// TwinCAT 3 PLC project RetentiveTimers
// Title: Retentive Timers
// Company: FisoThemes
// Author: Goodwill Mzumala
// ProjectVersion: 0.1.0.0
// Description: Standard library timers on TwinCAT count time by taking the difference between the current time from system timer and start time from system timer. While this is fine for most application, it is problematic for operations that require time to be retained even if the PLC is paused, stopped or turned off. For example, if a `TON` (Timer On-Delay) Timer is running and you stop the PLC Boot Project for a period of time, the `TON` will not resume from the point it was stopped. Instead it will skip time by the number of ms/secs/mins/hours it was stopped. This makes it useless for applications such as tracking the length of time a PLC has been running or retaining persistent time. Retentive variants of the Standard library timers stop this from happen. They are based on PLC Task cycle time rather than system time. This means they will simply stop counting when the PLC Task Cycle is stopped and will resume from where they left-off as soon as the task cycle picks up. All arguments behave in the same manner as those of the standard library.
// ProgramVersion: 3.1.4023.0
// libraries:
//   Tc2_Standard, * (Beckhoff Automation GmbH)
//   Tc2_System, * (Beckhoff Automation GmbH)
//   Tc3_Module, * (Beckhoff Automation GmbH)
// project tree:
//   DUTs/Structs/ ST_PLC_TASK_INFORMATION.TcDUT
//   / PlcTask.TcTTO
//   POUs/Examples/Section 1 - Standard Timers Comparisons/ P_Example_3_TPs.TcPOU, P_Section_1.TcPOU, P_Example_1_TONs.TcPOU, P_Example_2_TOFs.TcPOU
//   POUs/Examples/Section 2 - Pausable Timers Comparisons/ P_Section_2.TcPOU
//   POUs/Examples/Section 3 - Stopwatch/ P_Example_Stopwatch.TcPOU, P_Section_3.TcPOU
//   POUs/Function Blocks/ FB_RTimer.TcPOU, FB_RTON.TcPOU, FB_RTOF.TcPOU, FB_RTP.TcPOU, FB_RStopwatch.TcPOU, FB_Timer.TcPOU, FB_Stopwatch.TcPOU
//   POUs/Functions/ F_Get_PLC_Task_Information.TcPOU
//   POUs/ MAIN.TcPOU
// real-time tasks:
//   TASK PlcTask: cycle T#10ms, priority 20, ADS port 350

CONFIGURATION RetentiveTimers
    RESOURCE PLC ON TwinCAT3
        TASK PlcTask(INTERVAL := T#10ms, PRIORITY := 20);
        PROGRAM MAIN WITH PlcTask : MAIN;
    END_RESOURCE
END_CONFIGURATION

// ---- DUTs/Structs/ST_PLC_TASK_INFORMATION.TcDUT
TYPE ST_PLC_TASK_INFORMATION EXTENDS PlcTaskSystemInfo :
STRUCT
	tCycleTime 	: TIME; 	// Current task cycle time
	tlCycleTime : LTIME; 	// Current task cycle time in LTIME
END_STRUCT
END_TYPE

// ---- POUs/MAIN.TcPOU
PROGRAM MAIN
VAR
END_VAR

P_Section_1();
P_Section_2();
P_Section_3();

END_PROGRAM

// ---- POUs/Examples/Section 1 - Standard Timers Comparisons/P_Section_1.TcPOU
PROGRAM P_Section_1
VAR
END_VAR

P_Example_1_TONs();
P_Example_2_TOFs();
P_Example_3_TPs();

END_PROGRAM

// ---- POUs/Examples/Section 1 - Standard Timers Comparisons/P_Example_1_TONs.TcPOU
PROGRAM P_Example_1_TONs
VAR
	bStart 				: BOOL; 
	tSet_Time 			: TIME := T#10S; 
	tElapsed_Time_TON, 
	tElapsed_Time_RTON 	: TIME; 
	bElapsed_Time_TON,
	bElapsed_Time_RTON 	: BOOL; 
	
	fbTON 				: TON;
	fbRTON 				: FB_RTON;
	stPLC_Task_Info : ST_PLC_TASK_INFORMATION;
	nCC, nRCC 	: UDINT;
END_VAR

(*
NOTES:
	-> Activate Configuration and START(F5) PLC Boot Project
	-> Login (if you haven't already)
	-> Make sure both timers are set for 10 mins 
	-> Start the timers by writing a TRUE to the bStart variable
	-> Let the timers run for a little bit
	-> Notice that both elapsed time read are the same
	-> STOP(Shift+F5) the PLC Boot Project for approx. 10-30secs
	-> START(F5) the PLC Boot Project
	
	--> Notice the TON elapsed time (tElapsed_Time_TON) is 10-30secs ahead of the FB_RTON elapsed time (tElapsed_Time_RTON)
	--> FB_RTON resumes from where it left-off if PLC is stopped. 
*)

fbTON(IN := bStart, PT := tSet_Time, 
	  Q => bElapsed_Time_TON, ET => tElapsed_Time_TON);
	  
fbRTON(IN := bStart, PT := tSet_Time, 
	  Q => bElapsed_Time_RTON, ET => tElapsed_Time_RTON);

END_PROGRAM

// ---- POUs/Function Blocks/FB_RTON.TcPOU
(* Retentive Timer On-Delay - implements a timer-on delay that persists if PLC cycle is stopped. 
When the input gets TRUE, elapsed time ET will run until also the output Q becomes TRUE. 
*)
FUNCTION_BLOCK FB_RTON
VAR_INPUT
	IN 	: BOOL; // Starts timer with rising edge, resets timer with falling edge
	PT 	: TIME; // Time to pass, before Q is set
END_VAR
VAR_OUTPUT
	Q 	: BOOL; // Is TRUE, PT seconds after IN had a rising edge
	ET 	: TIME; // Elapsed time
END_VAR
VAR
	stPLC_Task_Info 	: ST_PLC_TASK_INFORMATION;
	tAccumulator 		: TIME;
	nLast_Cycle_Count 	: UDINT;
END_VAR

IF IN THEN
	stPLC_Task_Info := F_Get_PLC_Task_Information();
	Q := ET >= PT;
	
	IF NOT(Q) AND ((nLast_Cycle_Count <> stPLC_Task_Info.CycleCount) OR nLast_Cycle_Count = 0) THEN
		tAccumulator := tAccumulator + stPLC_Task_Info.tCycleTime; 
		ET := LIMIT(T#0MS, THIS^.Lerp(T#0MS, PT, TO_REAL(tAccumulator)/TO_REAL(PT))-stPLC_Task_Info.tCycleTime, PT);
		nLast_Cycle_Count := stPLC_Task_Info.CycleCount;
		END_IF
	RETURN;
	END_IF
tAccumulator := ET := T#0MS; Q := FALSE;

// Linear interpolation (Lerp) - this method interpolates values between 2 time points.
METHOD PRIVATE Lerp : TIME
VAR_INPUT
	tStart 	: TIME := T#0MS; 
	tFinish : TIME;
	fPercentage : REAL; // Value must be between 0 and 1
END_VAR
// Lerp(Start, Finish, Percentage) = Start + (Finish - Start)*Percentage
Lerp := TO_TIME(TO_REAL(tStart) + TO_REAL(tFinish - tStart)*fPercentage);
END_METHOD

END_FUNCTION_BLOCK

// ---- POUs/Functions/F_Get_PLC_Task_Information.TcPOU
(* Gets the infomation of the task the function is currently called on.
.. _More: https://infosys.beckhoff.com/english.php?content=../content/1033/globaldatatypes/714818699.html&id=
*)
FUNCTION F_Get_PLC_Task_Information : ST_PLC_TASK_INFORMATION
VAR_INPUT
END_VAR
VAR
	fbCurrent_Task_Index  	: GETCURTASKINDEX;
	st_TaskInfo 			: PlcTaskSystemInfo;
	stTask_Info 			: ST_PLC_TASK_INFORMATION;
END_VAR

fbCurrent_Task_Index();
st_TaskInfo 						:= TwinCAT_SystemInfoVarList._TaskInfo[fbCurrent_Task_Index.index];

stTask_Info.AdsPort 				:= st_TaskInfo.AdsPort;
stTask_Info.CycleCount 				:= st_TaskInfo.CycleCount;
stTask_Info.CycleTime 				:= st_TaskInfo.CycleTime;
stTask_Info.CycleTimeExceeded 		:= st_TaskInfo.CycleTimeExceeded;
stTask_Info.DcTaskTime 				:= st_TaskInfo.DcTaskTime;
stTask_Info.FirstCycle				:= st_TaskInfo.FirstCycle;
stTask_Info.InCallAfterOutputUpdate := st_TaskInfo.InCallAfterOutputUpdate;
stTask_Info.LastExecTime 			:= st_TaskInfo.LastExecTime;
stTask_Info.ObjId 					:= st_TaskInfo.ObjId;
stTask_Info.Priority 				:= st_TaskInfo.Priority;
stTask_Info.RTViolation 			:= st_TaskInfo.RTViolation;
stTask_Info.TaskName 				:= st_TaskInfo.TaskName;
stTask_Info.tlCycleTime 			:= TO_LTIME(st_TaskInfo.CycleTime*100);
stTask_Info.tCycleTime 				:= TO_TIME(stTask_Info.tlCycleTime);

F_Get_PLC_Task_Information 		:= stTask_Info;

END_FUNCTION

// ---- POUs/Examples/Section 1 - Standard Timers Comparisons/P_Example_2_TOFs.TcPOU
PROGRAM P_Example_2_TOFs
VAR
	bStart 				: BOOL; 
	tSet_Time 			: TIME := T#10S; 
	tElapsed_Time_TOF, 
	tElapsed_Time_RTOF 	: TIME; 
	bElapsed_Time_TOF,
	bElapsed_Time_RTOF 	: BOOL; 
	
	fbTOF 				: TOF;
	fbRTOF 				: FB_RTOF;
	
END_VAR

(*
NOTES:
	-> Activate Configuration and START(F5) PLC Boot Project
	-> Login (if you haven't already)
	-> Make sure both timers are set for 1 mins 
	-> Start the timers by writing a TRUE to the bStart variable
	-> Let the timers run for a little bit
	-> Notice that both elapsed time read are the same
	-> STOP(Shift+F5) the PLC Boot Project for approx. 10-30secs
	-> START(F5) the PLC Boot Project
	
	--> Notice the TOF elapsed time (tElapsed_Time_TOF) is 10-30secs ahead of the FB_RTOF elapsed time (tElapsed_Time_RTOF)
	--> FB_RTOF resumes from where it left-off if PLC is stopped. 
*)

fbTOF(IN := bStart, PT := tSet_Time, 
	  Q => bElapsed_Time_TOF, ET => tElapsed_Time_TOF);
	  
fbRTOF(IN := bStart, PT := tSet_Time, 
	  Q => bElapsed_Time_RTOF, ET => tElapsed_Time_RTOF);

END_PROGRAM

// ---- POUs/Function Blocks/FB_RTOF.TcPOU
(* Retentive Timer Off-Delay - implements a timer-off delay that persists if PLC cycle is stopped. 
When the input becomes FALSE after a TRUE, the elapsed time ET will run through until the output Q becomes TRUE. 
*)
FUNCTION_BLOCK FB_RTOF
VAR_INPUT
	IN 	: BOOL; // Starts timer with falling edge, resets timer with rising edge
	PT 	: TIME; // Time to pass, before Q is set
END_VAR
VAR_OUTPUT
	Q 	: BOOL; // is FALSE, PT seconds after IN had a falling edge
	ET 	: TIME; // Elapsed time
END_VAR
VAR
	stPLC_Task_Info 	: ST_PLC_TASK_INFORMATION;
	tAccumulator 		: TIME;
	nLast_Cycle_Count 	: UDINT;
	eState 				: (IDLE, RUN);
END_VAR

LBL_TOP: 
CASE eState OF
	IDLE: 
		IF IN THEN Q := TRUE; tAccumulator := ET := T#0MS; eState := RUN; JMP LBL_TOP; END_IF
	RUN:
		stPLC_Task_Info := F_Get_PLC_Task_Information();
		IF NOT(IN) AND ((nLast_Cycle_Count <> stPLC_Task_Info.CycleCount) OR nLast_Cycle_Count = 0) THEN 
			Q := ET <> PT;
			IF (ET >= PT) THEN Q := FALSE;  eState := IDLE; JMP LBL_TOP; END_IF
			tAccumulator := tAccumulator + stPLC_Task_Info.tCycleTime; 
			ET := LIMIT(T#0MS, THIS^.Lerp(T#0MS, PT, TO_REAL(tAccumulator)/TO_REAL(PT))-stPLC_Task_Info.tCycleTime, PT);
			END_IF
		nLast_Cycle_Count := stPLC_Task_Info.CycleCount;
		IF IN THEN tAccumulator := ET := T#0MS;END_IF
END_CASE

// Linear interpolation (Lerp) - this method interpolates values between 2 time points.
METHOD PRIVATE Lerp : TIME
VAR_INPUT
	tStart 	: TIME := T#0MS; 
	tFinish : TIME;
	fPercentage : REAL; // Value must be between 0 and 1
END_VAR
// Lerp(Start, Finish, Percentage) = Start + (Finish - Start)*Percentage
Lerp := TO_TIME(TO_REAL(tStart) + TO_REAL(tFinish - tStart)*fPercentage);
END_METHOD

END_FUNCTION_BLOCK

// ---- POUs/Examples/Section 1 - Standard Timers Comparisons/P_Example_3_TPs.TcPOU
PROGRAM P_Example_3_TPs
VAR
	bStart 				: BOOL; 
	tSet_Time 			: TIME := T#10S; 
	tElapsed_Time_TP, 
	tElapsed_Time_RTP 	: TIME; 
	bElapsed_Time_TP,
	bElapsed_Time_RTP 	: BOOL; 
	
	fbTP 				: TP;
	fbRTP 				: FB_RTP;
	
END_VAR

(*
NOTES:
	-> Activate Configuration and START(F5) PLC Boot Project
	-> Login (if you haven't already)
	-> Make sure both timers are set for 10 mins 
	-> Start the timers by writing a TRUE to the bStart variable
	-> Let the timers run for a little bit
	-> Notice that both elapsed time read are the same
	-> STOP(Shift+F5) the PLC Boot Project for approx. 10-30secs
	-> START(F5) the PLC Boot Project
	
	--> Notice the TP elapsed time (tElapsed_Time_TP) is 10-30secs ahead of the FB_RTOF elapsed time (tElapsed_Time_RTP)
	--> FB_RTP resumes from where it left-off if PLC is stopped. 
*)

fbTP(IN := bStart, PT := tSet_Time, 
	  Q => bElapsed_Time_TP, ET => tElapsed_Time_TP);
	  
fbRTP(IN := bStart, PT := tSet_Time, 
	  Q => bElapsed_Time_RTP, ET => tElapsed_Time_RTP);

END_PROGRAM

// ---- POUs/Function Blocks/FB_RTP.TcPOU
(* Retentive Pulse Timer - implements a pulse time that persists if PLC cycle is stopped. 
when the input becomes TRUE, the elapsed time ET will run for the set time PT and the output Q will becomes TRUE.  
*)
FUNCTION_BLOCK FB_RTP
VAR_INPUT
        IN      : BOOL; // Trigger for Start of the Signal
        PT      : TIME; // The length of the High-Signal in ms
END_VAR
VAR_OUTPUT
        Q       : BOOL; // The pulse
        ET      : TIME; // The current phase of the High-Signal
END_VAR
VAR
	stPLC_Task_Info 	: ST_PLC_TASK_INFORMATION;
	tAccumulator 		: TIME;
	nLast_Cycle_Count 	: UDINT;
	eState 				: (IDLE, RUN);
END_VAR

LBL_TOP:
CASE eState OF
	IDLE:
		tAccumulator := ET := T#0MS; Q := FALSE;
		IF IN THEN eState := RUN; JMP LBL_TOP; END_IF
	RUN:
		Q := ET < PT;
		IF (PT = t#0s) THEN RETURN; END_IF
		IF NOT(Q) AND NOT(IN) THEN eState := IDLE; JMP LBL_TOP; END_IF
		IF NOT(Q) THEN RETURN; END_IF
		stPLC_Task_Info := F_Get_PLC_Task_Information();
		IF (nLast_Cycle_Count = stPLC_Task_Info.CycleCount)THEN RETURN; END_IF
		tAccumulator := tAccumulator + stPLC_Task_Info.tCycleTime; 
		ET := LIMIT(T#0MS, THIS^.Lerp(T#0MS, PT, TO_REAL(tAccumulator)/TO_REAL(PT))-stPLC_Task_Info.tCycleTime, PT);
		nLast_Cycle_Count := stPLC_Task_Info.CycleCount;	
END_CASE

// Linear interpolation (Lerp) - this method interpolates values between 2 time points.
METHOD PRIVATE Lerp : TIME
VAR_INPUT
	tStart 	: TIME := T#0MS; 
	tFinish : TIME;
	fPercentage : REAL; // Value must be between 0 and 1
END_VAR
// Lerp(Start, Finish, Percentage) = Start + (Finish - Start)*Percentage
Lerp := TO_TIME(TO_REAL(tStart) + TO_REAL(tFinish - tStart)*fPercentage);
END_METHOD

END_FUNCTION_BLOCK

// ---- POUs/Examples/Section 2 - Pausable Timers Comparisons/P_Section_2.TcPOU
PROGRAM P_Section_2
VAR
	bStart, bPause 		: BOOL; 
	tSet_Time 			: TIME := T#10S; 
	tElapsed_Time,
	tElapsed_RTime 		: TIME; 
	bElapsed_Time,
	bElapsed_RTime 		: BOOL; 
	fbTimer 			: FB_Timer; 
	fbRTimer 			: FB_RTimer;
END_VAR

(*
NOTES:
	-> Activate Configuration and START(F5) PLC Boot Project
	-> Login (if you haven't already)
	-> Make sure both timers are set for 10 mins 
	-> Start the timers by writing a TRUE to the bStart variable
	-> Let the timers run for a little bit
	-> Notice that both elapsed time read are the same
	-> STOP(Shift+F5) the PLC Boot Project for approx. 10-30secs
	-> START(F5) the PLC Boot Project
	
	--> Notice the FB_Timer's elapsed time (tElapsed_Time) is 10-30secs ahead of the FB_RTimer's elapsed time (tElapsed_RTime)
	--> FB_RTimer resumes from where it left-off if PLC is stopped. 
*)

fbTimer(bStart := bStart, bPause := bPause, tSet := tSet_Time, 
		bElapsed => bElapsed_Time, tElapsed => tElapsed_Time);
fbRTimer(bStart := bStart, bPause := bPause, tSet := tSet_Time,  
		 bElapsed => bElapsed_RTime, tElapsed => tElapsed_RTime);

END_PROGRAM

// ---- POUs/Function Blocks/FB_Timer.TcPOU
// Pausable Timer Function Block
FUNCTION_BLOCK FB_Timer
VAR_INPUT
    bStart 		: BOOL; // Start (TRUE) or Stop (FALSE) Timer 
	bPause 		: BOOL; // Pause Timer (TRUE), Only Pauses if IN := TRUE
    tSet		: TIME; // Set Time
END_VAR
VAR_OUTPUT
    bElapsed 	: BOOL;	// Becomes TRUE after Set Time has passed
    tElapsed 	: TIME; // Time Elapsed
END_VAR
VAR
	fbTON 		: TON;
	tPaused 	: TIME;
	eState		: (START, PAUSE);
END_VAR

IF NOT(bStart) THEN tPaused := tElapsed := T#0MS; END_IF
fbTON(PT := tSet - tPaused, Q => bElapsed);
IF bPause THEN 
	tPaused := fbTON.ET + tPaused; 
	fbTON(IN := FALSE); 
ELSE 
	fbTON(IN := bStart); 
	tElapsed := fbTON.ET + tPaused; 
	END_IF

END_FUNCTION_BLOCK

// ---- POUs/Function Blocks/FB_RTimer.TcPOU
// Retentive Pausable Timer Function Block
FUNCTION_BLOCK FB_RTimer
VAR_INPUT
    bStart 		: BOOL; // Start (TRUE) or Stop (FALSE) Timer 
	bPause 		: BOOL; // Pause Timer (TRUE), Only Pauses if IN := TRUE
    tSet		: TIME; // Set Time
END_VAR
VAR_OUTPUT
    bElapsed 	: BOOL;	// Becomes TRUE after Set Time has passed
    tElapsed 	: TIME; // Time Elapsed
END_VAR
VAR
	fbRTON 		: FB_RTON;
END_VAR

IF NOT(bStart) THEN fbRTON(IN := FALSE, Q => bElapsed, ET => tElapsed); RETURN; END_IF
IF bPause THEN RETURN; END_IF;
fbRTON(IN := TRUE, PT := tSet, Q => bElapsed, ET => tElapsed);

END_FUNCTION_BLOCK

// ---- POUs/Examples/Section 3 - Stopwatch/P_Section_3.TcPOU
PROGRAM P_Section_3
VAR
END_VAR

P_Example_Stopwatch();

END_PROGRAM

// ---- POUs/Examples/Section 3 - Stopwatch/P_Example_Stopwatch.TcPOU
PROGRAM P_Example_Stopwatch
VAR
	bStart 						: BOOL; 
	tElapsed_Time_Stopwatch, 
	tElapsed_Time_RStopwatch 	: TIME; 
	fbStopwatch 				: FB_Stopwatch;
	fbRStopwatch 				: FB_RStopwatch;
END_VAR

(*
NOTES:
	-> Activate Configuration and START(F5) PLC Boot Project
	-> Login (if you haven't already)
	-> Make sure both timers are set for 10 mins 
	-> Start the timers by writing a TRUE to the bStart variable
	-> Let the timers run for a little bit
	-> Notice that both elapsed time read are the same
	-> STOP(Shift+F5) the PLC Boot Project for approx. 10-30secs
	-> START(F5) the PLC Boot Project
*)

fbStopwatch(bStart := bStart, tElapsed => tElapsed_Time_Stopwatch);
fbRStopwatch(bStart := bStart, tElapsed => tElapsed_Time_RStopwatch);

END_PROGRAM

// ---- POUs/Function Blocks/FB_Stopwatch.TcPOU
FUNCTION_BLOCK FB_Stopwatch
VAR_INPUT
	bStart : BOOL;
END_VAR
VAR_OUTPUT
	tElapsed : TIME;
END_VAR
VAR
	stPLC_Task_Info : ST_PLC_TASK_INFORMATION;
	tAccumilator 	: TIME;
	fbTON 			: TON;
END_VAR

IF bStart THEN stPLC_Task_Info := F_Get_PLC_Task_Information(); END_IF
fbTON(PT := stPLC_Task_Info.tCycleTime*2 + tAccumilator);
fbTON(IN := bStart AND NOT(fbTON.Q));
tAccumilator := fbTON.ET; 
IF bStart THEN tElapsed := tAccumilator; END_IF

END_FUNCTION_BLOCK

// ---- POUs/Function Blocks/FB_RStopwatch.TcPOU
// Retentive stopwatch
FUNCTION_BLOCK FB_RStopwatch
VAR_INPUT
	bStart : BOOL;
END_VAR
VAR_OUTPUT
	tElapsed : TIME;
END_VAR
VAR
	stPLC_Task_Info : ST_PLC_TASK_INFORMATION;
	tAccumilator 	: TIME;
	fbTON 			: FB_RTON;
END_VAR

IF bStart THEN stPLC_Task_Info := F_Get_PLC_Task_Information(); END_IF
fbTON(PT := stPLC_Task_Info.tCycleTime*2 + tAccumilator);
fbTON(IN := bStart AND NOT(fbTON.Q));
tAccumilator := fbTON.ET; 
IF bStart THEN tElapsed := tAccumilator; END_IF

END_FUNCTION_BLOCK
